// LS Electric XG5000 project: motor
// PLC LSPLC
// module base 0 slot 0: 입출력 모듈:XBC-DR14E (DC 24V 입력 8점, 릴레이 출력 6점)

PROGRAM NewProgram (task: 스캔 프로그램)

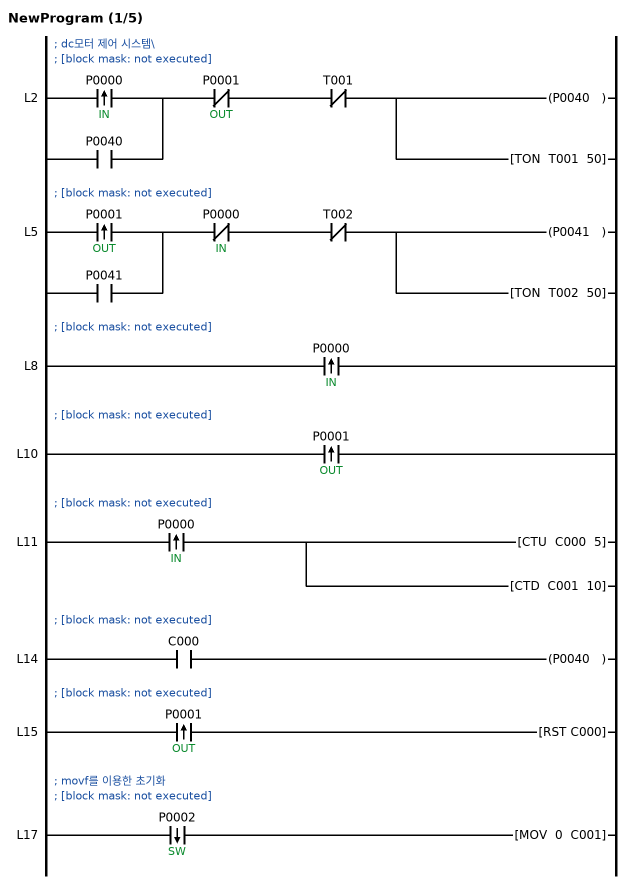
// dc모터 제어 시스템\
; L2 (block mask: not executed)
LOADP     P0000	// IN
OR        P0040
AND NOT   P0001	// OUT
AND NOT   T001
OUT       P0040
TON       T001 50
; L5 (block mask: not executed)
LOADP     P0001	// OUT
OR        P0041
AND NOT   P0000	// IN
AND NOT   T002
OUT       P0041
TON       T002 50
; L8 (block mask: not executed)
LOADP     P0000	// IN
; L10 (block mask: not executed)
LOADP     P0001	// OUT
; L11 (block mask: not executed)
LOADP     P0000	// IN
CTU       C000 5
CTD       C001 10
; L14 (block mask: not executed)
LOAD      C000
OUT       P0040
; L15 (block mask: not executed)
LOADP     P0001	// OUT
RST       C000
// movf를 이용한 초기화
; L17 (block mask: not executed)
LOADN     P0002	// SW
MOV       0 C001

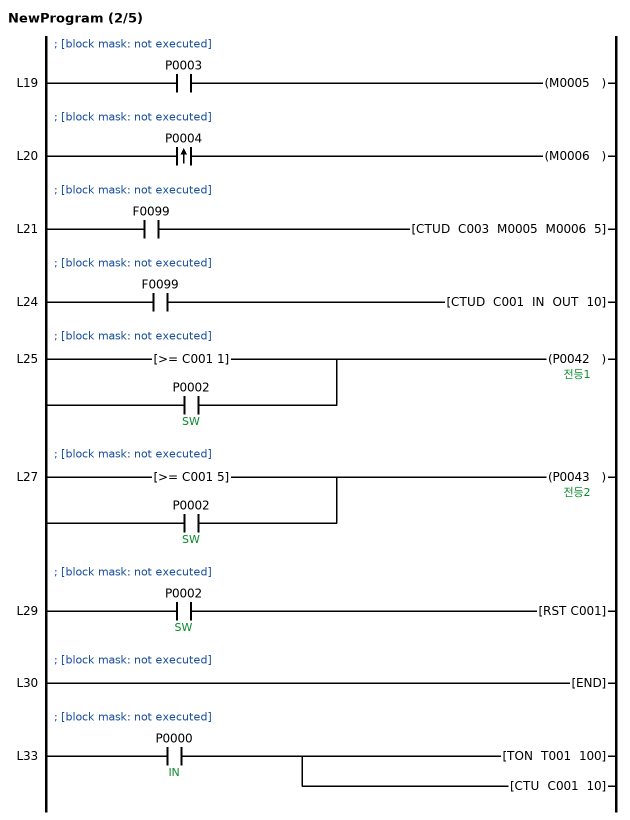
; L19 (block mask: not executed)
LOAD      P0003
OUT       M0005
; L20 (block mask: not executed)
LOADP     P0004
OUT       M0006
; L21 (block mask: not executed)
LOAD      F0099
CTUD      C003 M0005 M0006 5
; L24 (block mask: not executed)
LOAD      F0099
CTUD      C001 IN OUT 10
; L25 (block mask: not executed)
LOAD>=    C001 1
OR        P0002	// SW
OUT       P0042	// 전등1
; L27 (block mask: not executed)
LOAD>=    C001 5
OR        P0002	// SW
OUT       P0043	// 전등2
; L29 (block mask: not executed)
LOAD      P0002	// SW
RST       C001
; L30 (block mask: not executed)
END
; L33 (block mask: not executed)
LOAD      P0000	// IN
TON       T001 100
CTU       C001 10

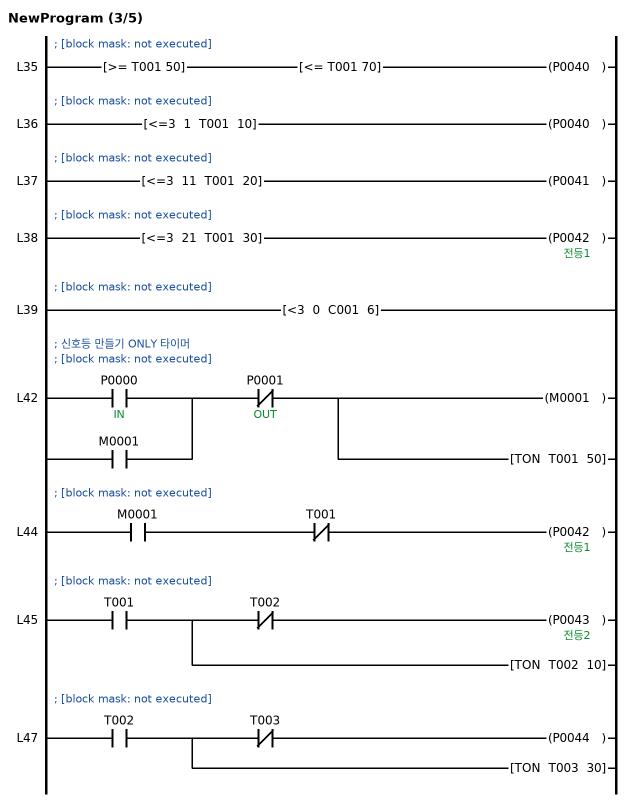
; L35 (block mask: not executed)
LOAD>=    T001 50
AND<=     T001 70
OUT       P0040
; L36 (block mask: not executed)
LOAD<=3   1 T001 10
OUT       P0040
; L37 (block mask: not executed)
LOAD<=3   11 T001 20
OUT       P0041
; L38 (block mask: not executed)
LOAD<=3   21 T001 30
OUT       P0042	// 전등1
; L39 (block mask: not executed)
LOAD<3    0 C001 6
// 신호등 만들기 ONLY 타이머
; L42 (block mask: not executed)
LOAD      P0000	// IN
OR        M0001
AND NOT   P0001	// OUT
OUT       M0001
TON       T001 50
; L44 (block mask: not executed)
LOAD      M0001
AND NOT   T001
OUT       P0042	// 전등1
; L45 (block mask: not executed)
LOAD      T001
MPUSH
AND NOT   T002
OUT       P0043	// 전등2
MPOP
TON       T002 10
; L47 (block mask: not executed)
LOAD      T002
MPUSH
AND NOT   T003
OUT       P0044
MPOP
TON       T003 30

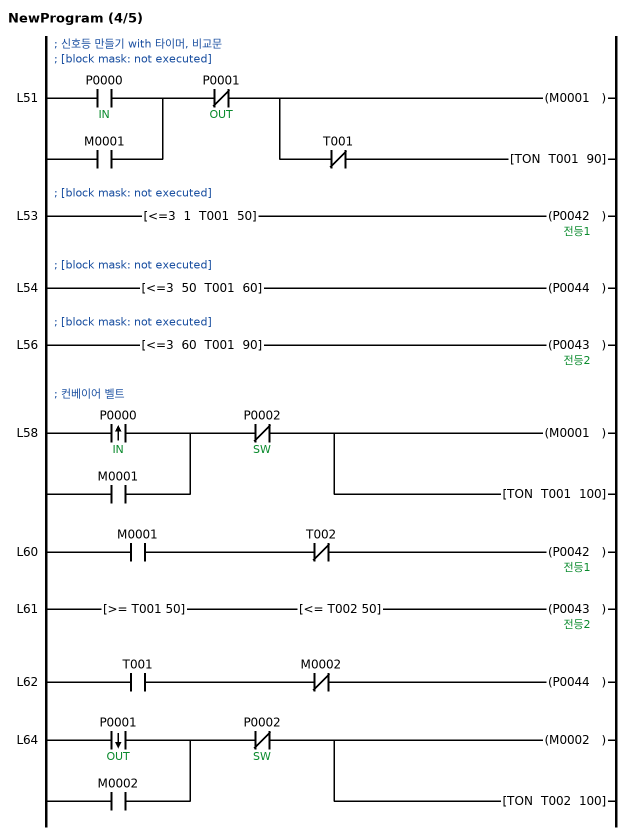
// 신호등 만들기 with 타이머, 비교문
; L51 (block mask: not executed)
LOAD      P0000	// IN
OR        M0001
AND NOT   P0001	// OUT
OUT       M0001
AND NOT   T001
TON       T001 90
; L53 (block mask: not executed)
LOAD<=3   1 T001 50
OUT       P0042	// 전등1
; L54 (block mask: not executed)
LOAD<=3   50 T001 60
OUT       P0044
; L56 (block mask: not executed)
LOAD<=3   60 T001 90
OUT       P0043	// 전등2
// 컨베이어 벨트
; L58
LOADP     P0000	// IN
OR        M0001
AND NOT   P0002	// SW
OUT       M0001
TON       T001 100
; L60
LOAD      M0001
AND NOT   T002
OUT       P0042	// 전등1
; L61
LOAD>=    T001 50
AND<=     T002 50
OUT       P0043	// 전등2
; L62
LOAD      T001
AND NOT   M0002
OUT       P0044
; L64
LOADN     P0001	// OUT
OR        M0002
AND NOT   P0002	// SW
OUT       M0002
TON       T002 100

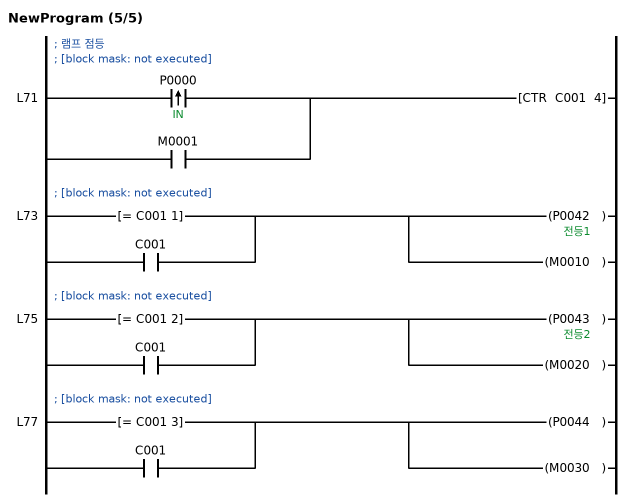
// 램프 점등
; L71 (block mask: not executed)
LOADP     P0000	// IN
OR        M0001
CTR       C001 4
; L73 (block mask: not executed)
LOAD=     C001 1
OR        C001
OUT       P0042	// 전등1
OUT       M0010
; L75 (block mask: not executed)
LOAD=     C001 2
OR        C001
OUT       P0043	// 전등2
OUT       M0020
; L77 (block mask: not executed)
LOAD=     C001 3
OR        C001
OUT       P0044
OUT       M0030